(* Logix 5000 project; controller GitProgram vendor 1 type 14 code 164 rev 30.11; software revision 30.00 *)
// This is a program used in the test of git.

TASK MainTask (continuous, watchdog 500 ms) : MainProgram

MODULES
   Local : vendor 1 type 14 code 164 (ICP 0, rev 30.11)
END_MODULES

VAR_GLOBAL   (* controller tags *)
   Calibrated_Level : DINT;
   Calibrated_Pressure : DINT;
   Calibrated_Pressure2 : DINT;
   Calibrated_Temperature : DINT;
   Calibrated_weight : DINT;
   Level : DINT;
   Offser : DINT := 30;
   Offset : DINT := 20;
   Pressure : DINT := 130;
   Pressure2 : DINT;
   Temperature : DINT := 155;
   weight : DINT;
END_VAR

PROGRAM MainProgram   (* main routine MainRoutine *)

ROUTINE MainRoutine   (* ladder *)
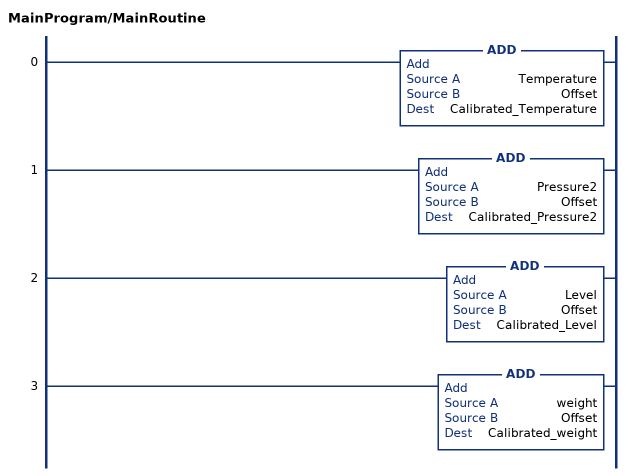
   0: ADD(Temperature,Offset,Calibrated_Temperature);
   1: ADD(Pressure2,Offset,Calibrated_Pressure2);
   2: ADD(Level,Offset,Calibrated_Level);
   3: ADD(weight,Offset,Calibrated_weight);
END_ROUTINE
END_PROGRAM
